Omron CX-Programmer project NewProject (CX-Programmer 9.73)

# PLC PLCMIX: CP1H XA

## Global symbols (name address type ; comment)
0.05 BOOL  ; PROXB
0.06 BOOL  ; PROXU
0.07 BOOL  ; PROXD
100.00 BOOL  ; WATER PUMP
100.01 BOOL  ; OIL PUMP
100.02 BOOL  ; VACUUM PUMP
100.03 BOOL  ; VACUUM RELEASE
100.04 BOOL  ; WATER HEATER
100.05 BOOL  ; VALVE UP
100.06 BOOL  ; VALVE DOWN
100.07 BOOL  ; UP MAX
100.08 BOOL  ; DOWN MAX
100.09 BOOL  ; POS BOWL
100.10 BOOL  ; UPPER LIMIT
100.11 BOOL  ; A
100.12 BOOL  ; UNDER LIMIT
100.13 BOOL  ; B
100.14 BOOL  ; ALARM WT TEMP
100.15 BOOL  ; ALARM MT TEMP
101.00 BOOL  ; CW
101.01 BOOL  ; CCW
101.02 BOOL  ; MAIN TIMER
101.03 BOOL  ; VALVE CW
101.04 BOOL  ; VALVE CCW
101.05 BOOL  ; ALARM LP
101.06 BOOL  ; DATA LOG
101.07 BOOL  ; ALARM TOR
10.00 BOOL  ; FLAG CALCULATE
200 CHANNEL  ; OPRESS
201 CHANNEL  ; VPRESS
2013 CHANNEL  ; RWT RAW VALUE
2014 CHANNEL  ; RWT RAW VALUE
2023 CHANNEL  ; ROT RAW VALUE
210 CHANNEL  ; DA FREQUENCY
300 CHANNEL  ; TIMER CW
301 CHANNEL  ; TIMER CCW
302 CHANNEL  ; MAIN TIMER
50.00 BOOL  ; UNDER LIMIT OPRESS
50.01 BOOL  ; UPPER LIMIT OPRESS
50.02 BOOL  ; UNDER LIMIT VPRESS
50.03 BOOL  ; UPPER LIMIT VPRESS
C0000 BOOL  ; COUNTER 1 WP
C0001 BOOL  ; COUNTER 2 WP
C0002 BOOL  ; COUNTER 1 OP
C0003 BOOL  ; COUNTER 2 OP
C0004 BOOL  ; COUNTER 1 VP
C0005 BOOL  ; COUNTER 2 VP
C0006 BOOL  ; COUNTER 1 WH
C0007 BOOL  ; COUNTER 2 WH
C0008 BOOL  ; Counter 1 UP
C0009 BOOL  ; Counter 2 UP
C0010 BOOL  ; Counter 1 DOWN
C0011 BOOL  ; Counter 2 DOWN
D0 CHANNEL  ; VALUE DA FREQUENCY
D1 CHANNEL  ; TOTAL BIT DA FREQUENCY
D10 CHANNEL  ; RWT MOV TO D10
D100 CHANNEL  ; INPUT SET MINUTE MTIM
D101 CHANNEL  ; MINUTE MTIM
D102 CHANNEL  ; INPUT SET SECOND MTIM
D103 CHANNEL  ; SECOND MTIM
D104 CHANNEL  ; INPUT SET MINUTE DIRTIM
D105 CHANNEL  ; MINUTE DIRTIM
D106 CHANNEL  ; INPUT SET SECOND DIRTIM
D107 CHANNEL  ; SECOND DIRITM
D11 CHANNEL  ; RMT MOV TO D11
D110 CHANNEL  ; MINUTE TO SECOND MTIM
D112 CHANNEL  ; SECOND TO SECOND MTIM
D114 CHANNEL  ; TOTAL SECOND MTIM
D116 CHANNEL  ; MINUTE TO SECOND DIRTIM
D118 CHANNEL  ; SECOND TO SECOND DIRTIM
D12 CHANNEL  ; ROT MOV TO D12
D120 CHANNEL  ; TOTAL SECOND DIRTIM
D130 CHANNEL  ; PV TIMER CW
D132 CHANNEL  ; PV TIMER CCW
D134 CHANNEL  ; PV MAIN TIMER
D136 CHANNEL  ; REAL SECOND
D140 CHANNEL  ; SECOND BCD TO CLOCK
D142 CHANNEL  ; SECOND DISPLAY
D144 CHANNEL  ; MINUTE DISPLAY
D146 CHANNEL  ; SET LP
D148 CHANNEL  ; DIVISOR KPA TO MPA
D150 CHANNEL  ; CONSTANTA PRES TO TORQUE
D152 CHANNEL  ; OPRESS KPA TO MPA
D154 CHANNEL  ; TORQUE RTOR NM
D156 CHANNEL  ; BACK TO NULL
D158 CHANNEL  ; SET TOR
D20 CHANNEL  ; RWT REAL NUM
D22 CHANNEL  ; RMT REAL NUM
D24 CHANNEL  ; ROT REAL NUM
D26 CHANNEL  ; DIVISOR WORD
D30 CHANNEL  ; RWT TEMP
D32 CHANNEL  ; RMT TEMP
D34 CHANNEL  ; ROT TEMP
D40 CHANNEL  ; SET WT TEMP
D42 CHANNEL  ; SET MT TEMP
D50 CHANNEL  ; RAW AD OPRESS
D51 CHANNEL  ; RAW AD VPRESS
D52 CHANNEL  ; MIN RANGE PRESSURE OPRESS
D54 CHANNEL  ; MAX RANGE PRESSURE OPRESS
D55 CHANNEL  ; MAX RANGE BIT
D56 CHANNEL  ; RESULTS SCL OPRESS
D57 CHANNEL  ; BIN OPRESS
D60 CHANNEL  ; MIN RANGE PRESSURE VPRESS
D62 CHANNEL  ; MAX RANGE PRESSURE VPRESS
D63 CHANNEL  ; MAX RANGE BIT
D64 CHANNEL  ; RESULTS SCL VPRESS
D65 CHANNEL  ; BIN VPRESS
D66 CHANNEL  ; DIVISOR 10
D68 CHANNEL  ; FLT OPRESS
D70 CHANNEL  ; FLT VPRESS
D72 CHANNEL  ; OPRESS (BAR UNIT)
D74 CHANNEL  ; BAR TO KPA
D76 CHANNEL  ; OPRESS (KPA UNIT)
D80 CHANNEL  ; MULTIPLY MBAR TO KPA
D82 CHANNEL  ; VPRESS (MBAR UNIT)
D84 CHANNEL  ; VPRESS (KPA UNIT)
D86 CHANNEL  ; PV ENCODER
D88 CHANNEL  ; FLT PV ENCODER
D90 CHANNEL  ; FLT MULTIPLY 60
D92 CHANNEL  ; FLT DIVISOR 2000
D94 CHANNEL  ; PV ENCODER MULTIPLY 60
D96 CHANNEL  ; RPM
W0.00 BOOL  ; PB WP
W0.01 BOOL  ; PB OP
W0.02 BOOL  ; PB VP
W0.03 BOOL  ; PB VR
W0.04 BOOL  ; PB WH
W0.05 BOOL  ; PB UP
W0.06 BOOL  ; PB DOWN
W0.07 BOOL  ; PB FAST
W0.08 BOOL  ; PB SLOW
W0.09 BOOL  ; SET TIME
W0.10 BOOL  ; CW
W0.11 BOOL  ; CCW
W0.12 BOOL  ; PROSES
W0.13 BOOL  ; STOP

## Program NewProgram1 (cyclic task 0)

### Section Section1

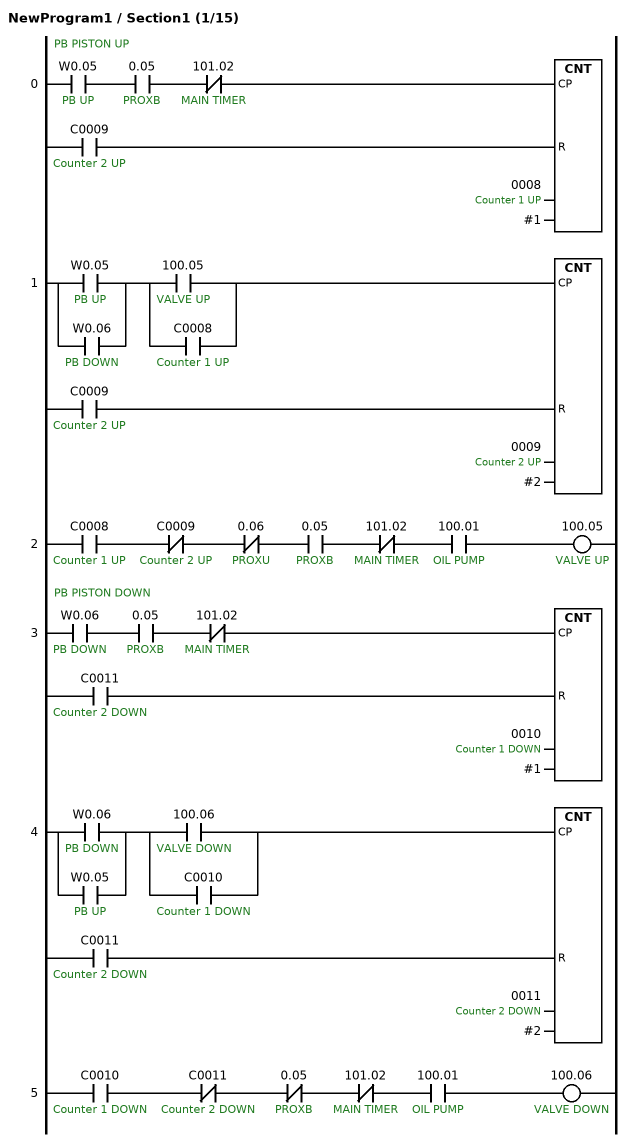
; rung 0: PB PISTON UP
LD W0.05  ; PB UP
AND 0.05  ; PROXB
ANDNOT 101.02  ; MAIN TIMER
LD C0009  ; Counter 2 UP
CNT 0008 #1  ; Counter 1 UP
; rung 1
LD W0.05  ; PB UP
OR W0.06  ; PB DOWN
LD 100.05  ; VALVE UP
OR C0008  ; Counter 1 UP
ANDLD
LD C0009  ; Counter 2 UP
CNT 0009 #2  ; Counter 2 UP
; rung 2
LD C0008  ; Counter 1 UP
ANDNOT C0009  ; Counter 2 UP
ANDNOT 0.06  ; PROXU
AND 0.05  ; PROXB
ANDNOT 101.02  ; MAIN TIMER
AND 100.01  ; OIL PUMP
OUT 100.05  ; VALVE UP
; rung 3: PB PISTON DOWN
LD W0.06  ; PB DOWN
AND 0.05  ; PROXB
ANDNOT 101.02  ; MAIN TIMER
LD C0011  ; Counter 2 DOWN
CNT 0010 #1  ; Counter 1 DOWN
; rung 4
LD W0.06  ; PB DOWN
OR W0.05  ; PB UP
LD 100.06  ; VALVE DOWN
OR C0010  ; Counter 1 DOWN
ANDLD
LD C0011  ; Counter 2 DOWN
CNT 0011 #2  ; Counter 2 DOWN
; rung 5
LD C0010  ; Counter 1 DOWN
ANDNOT C0011  ; Counter 2 DOWN
ANDNOT 0.05  ; PROXB
ANDNOT 101.02  ; MAIN TIMER
AND 100.01  ; OIL PUMP
OUT 100.06  ; VALVE DOWN

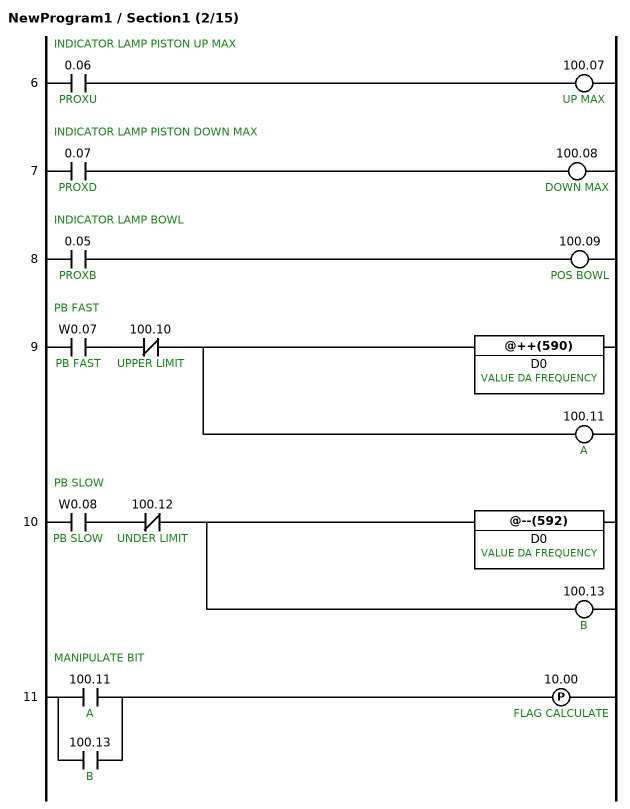
; rung 6: INDICATOR LAMP PISTON UP MAX
LD 0.06  ; PROXU
OUT 100.07  ; UP MAX
; rung 7: INDICATOR LAMP PISTON DOWN MAX
LD 0.07  ; PROXD
OUT 100.08  ; DOWN MAX
; rung 8: INDICATOR LAMP BOWL
LD 0.05  ; PROXB
OUT 100.09  ; POS BOWL
; rung 9: PB FAST
LD W0.07  ; PB FAST
ANDNOT 100.10  ; UPPER LIMIT
@++(590) D0  ; VALUE DA FREQUENCY
OUT 100.11  ; A
; rung 10: PB SLOW
LD W0.08  ; PB SLOW
ANDNOT 100.12  ; UNDER LIMIT
@--(592) D0  ; VALUE DA FREQUENCY
OUT 100.13  ; B
; rung 11: MANIPULATE BIT
LD 100.11  ; A
OR 100.13  ; B
DIFU(013) 10.00  ; FLAG CALCULATE

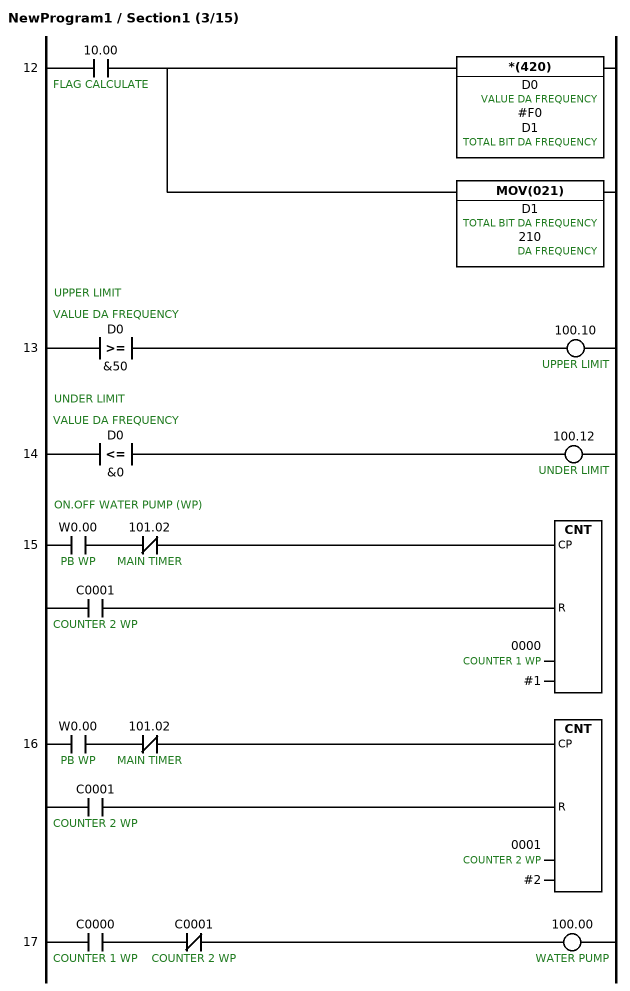
; rung 12
LD 10.00  ; FLAG CALCULATE
*(420) D0 #F0 D1  ; VALUE DA FREQUENCY, TOTAL BIT DA FREQUENCY
MOV(021) D1 210  ; TOTAL BIT DA FREQUENCY, DA FREQUENCY
; rung 13: UPPER LIMIT
LD>=(325) D0 &50  ; VALUE DA FREQUENCY
OUT 100.10  ; UPPER LIMIT
; rung 14: UNDER LIMIT
LD<=(315) D0 &0  ; VALUE DA FREQUENCY
OUT 100.12  ; UNDER LIMIT
; rung 15: ON.OFF WATER PUMP (WP)
LD W0.00  ; PB WP
ANDNOT 101.02  ; MAIN TIMER
LD C0001  ; COUNTER 2 WP
CNT 0000 #1  ; COUNTER 1 WP
; rung 16
LD W0.00  ; PB WP
ANDNOT 101.02  ; MAIN TIMER
LD C0001  ; COUNTER 2 WP
CNT 0001 #2  ; COUNTER 2 WP
; rung 17
LD C0000  ; COUNTER 1 WP
ANDNOT C0001  ; COUNTER 2 WP
OUT 100.00  ; WATER PUMP

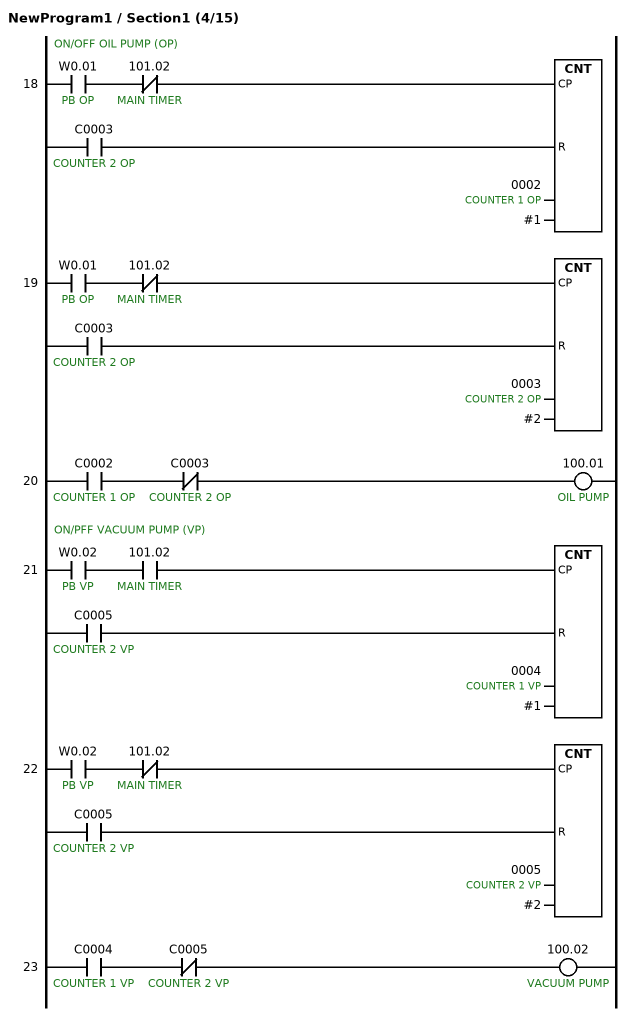
; rung 18: ON/OFF OIL PUMP (OP)
LD W0.01  ; PB OP
ANDNOT 101.02  ; MAIN TIMER
LD C0003  ; COUNTER 2 OP
CNT 0002 #1  ; COUNTER 1 OP
; rung 19
LD W0.01  ; PB OP
ANDNOT 101.02  ; MAIN TIMER
LD C0003  ; COUNTER 2 OP
CNT 0003 #2  ; COUNTER 2 OP
; rung 20
LD C0002  ; COUNTER 1 OP
ANDNOT C0003  ; COUNTER 2 OP
OUT 100.01  ; OIL PUMP
; rung 21: ON/PFF VACUUM PUMP (VP)
LD W0.02  ; PB VP
AND 101.02  ; MAIN TIMER
LD C0005  ; COUNTER 2 VP
CNT 0004 #1  ; COUNTER 1 VP
; rung 22
LD W0.02  ; PB VP
ANDNOT 101.02  ; MAIN TIMER
LD C0005  ; COUNTER 2 VP
CNT 0005 #2  ; COUNTER 2 VP
; rung 23
LD C0004  ; COUNTER 1 VP
ANDNOT C0005  ; COUNTER 2 VP
OUT 100.02  ; VACUUM PUMP

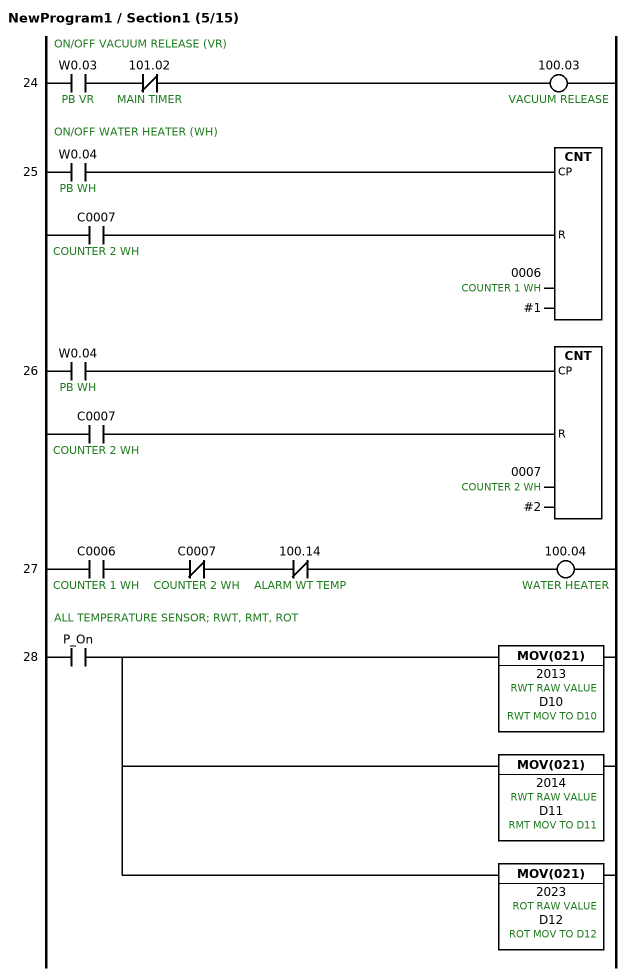
; rung 24: ON/OFF VACUUM RELEASE (VR)
LD W0.03  ; PB VR
ANDNOT 101.02  ; MAIN TIMER
OUT 100.03  ; VACUUM RELEASE
; rung 25: ON/OFF WATER HEATER (WH)
LD W0.04  ; PB WH
LD C0007  ; COUNTER 2 WH
CNT 0006 #1  ; COUNTER 1 WH
; rung 26
LD W0.04  ; PB WH
LD C0007  ; COUNTER 2 WH
CNT 0007 #2  ; COUNTER 2 WH
; rung 27
LD C0006  ; COUNTER 1 WH
ANDNOT C0007  ; COUNTER 2 WH
ANDNOT 100.14  ; ALARM WT TEMP
OUT 100.04  ; WATER HEATER
; rung 28: ALL TEMPERATURE SENSOR; RWT, RMT, ROT
LD P_On
MOV(021) 2013 D10  ; RWT RAW VALUE, RWT MOV TO D10
MOV(021) 2014 D11  ; RWT RAW VALUE, RMT MOV TO D11
MOV(021) 2023 D12  ; ROT RAW VALUE, ROT MOV TO D12

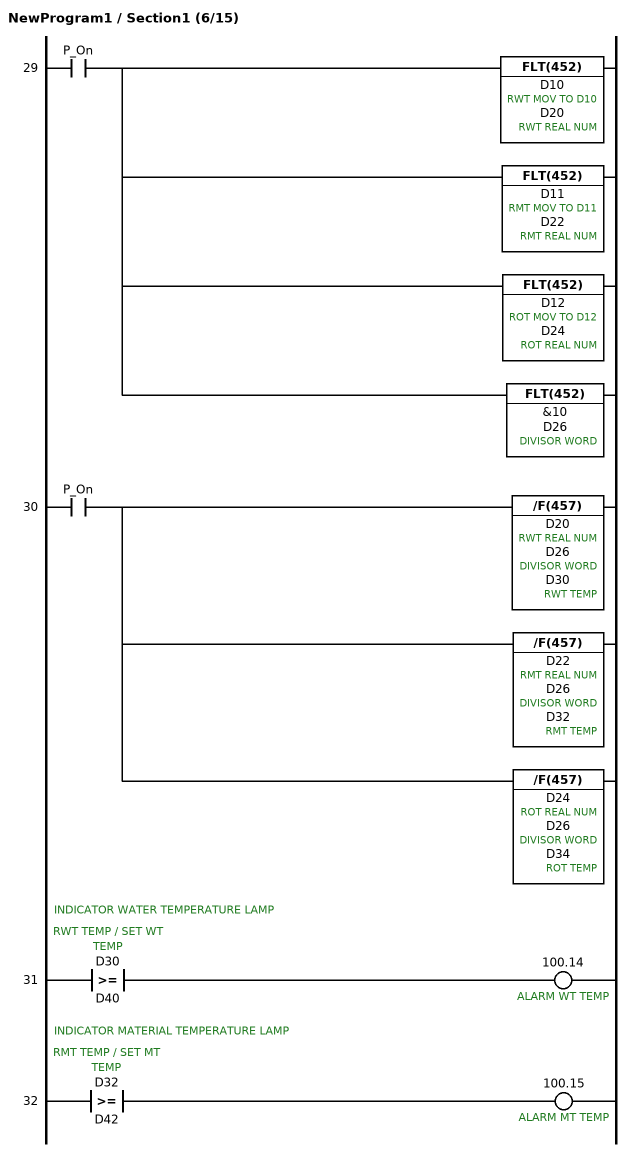
; rung 29
LD P_On
FLT(452) D10 D20  ; RWT MOV TO D10, RWT REAL NUM
FLT(452) D11 D22  ; RMT MOV TO D11, RMT REAL NUM
FLT(452) D12 D24  ; ROT MOV TO D12, ROT REAL NUM
FLT(452) &10 D26  ; DIVISOR WORD
; rung 30
LD P_On
/F(457) D20 D26 D30  ; RWT REAL NUM, DIVISOR WORD, RWT TEMP
/F(457) D22 D26 D32  ; RMT REAL NUM, DIVISOR WORD, RMT TEMP
/F(457) D24 D26 D34  ; ROT REAL NUM, DIVISOR WORD, ROT TEMP
; rung 31: INDICATOR WATER TEMPERATURE LAMP
LD>=F(334) D30 D40  ; RWT TEMP, SET WT TEMP
OUT 100.14  ; ALARM WT TEMP
; rung 32: INDICATOR MATERIAL TEMPERATURE LAMP
LD>=F(334) D32 D42  ; RMT TEMP, SET MT TEMP
OUT 100.15  ; ALARM MT TEMP

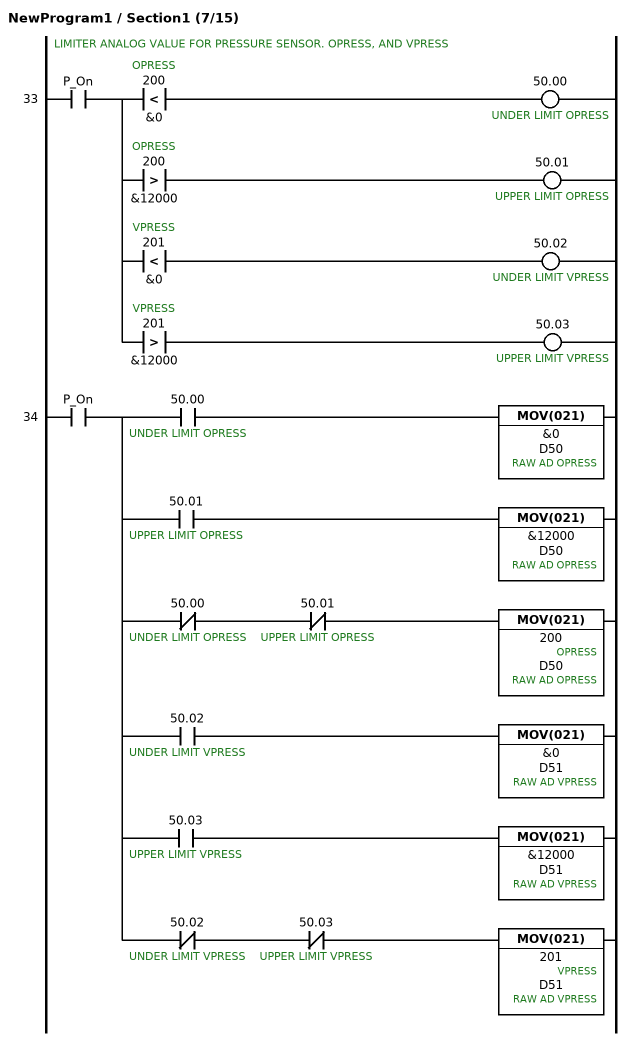
; rung 33: LIMITER ANALOG VALUE FOR PRESSURE SENSOR. OPRESS, AND VPRESS
LD P_On
OUT TR0
AND<S(312) 200 &0  ; OPRESS
OUT 50.00  ; UNDER LIMIT OPRESS
LD TR0
AND>S(322) 200 &12000  ; OPRESS
OUT 50.01  ; UPPER LIMIT OPRESS
LD TR0
AND<S(312) 201 &0  ; VPRESS
OUT 50.02  ; UNDER LIMIT VPRESS
LD TR0
AND>S(322) 201 &12000  ; VPRESS
OUT 50.03  ; UPPER LIMIT VPRESS
; rung 34
LD P_On
OUT TR0
AND 50.00  ; UNDER LIMIT OPRESS
MOV(021) &0 D50  ; RAW AD OPRESS
LD TR0
AND 50.01  ; UPPER LIMIT OPRESS
MOV(021) &12000 D50  ; RAW AD OPRESS
LD TR0
ANDNOT 50.00  ; UNDER LIMIT OPRESS
ANDNOT 50.01  ; UPPER LIMIT OPRESS
MOV(021) 200 D50  ; OPRESS, RAW AD OPRESS
LD TR0
AND 50.02  ; UNDER LIMIT VPRESS
MOV(021) &0 D51  ; RAW AD VPRESS
LD TR0
AND 50.03  ; UPPER LIMIT VPRESS
MOV(021) &12000 D51  ; RAW AD VPRESS
LD TR0
ANDNOT 50.02  ; UNDER LIMIT VPRESS
ANDNOT 50.03  ; UPPER LIMIT VPRESS
MOV(021) 201 D51  ; VPRESS, RAW AD VPRESS

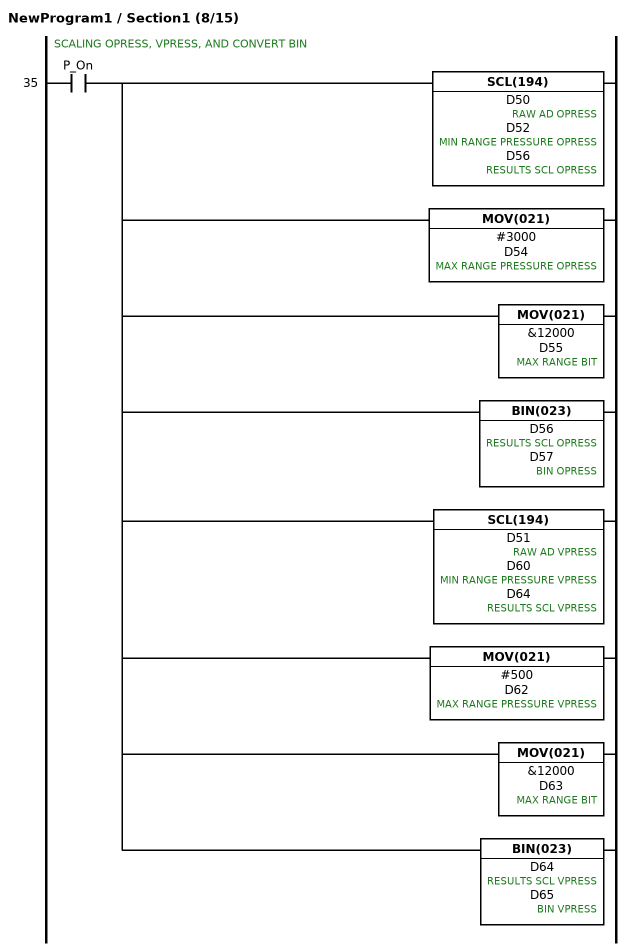
; rung 35: SCALING OPRESS, VPRESS, AND CONVERT BIN
LD P_On
SCL(194) D50 D52 D56  ; RAW AD OPRESS, MIN RANGE PRESSURE OPRESS, RESULTS SCL OPRESS
MOV(021) #3000 D54  ; MAX RANGE PRESSURE OPRESS
MOV(021) &12000 D55  ; MAX RANGE BIT
BIN(023) D56 D57  ; RESULTS SCL OPRESS, BIN OPRESS
SCL(194) D51 D60 D64  ; RAW AD VPRESS, MIN RANGE PRESSURE VPRESS, RESULTS SCL VPRESS
MOV(021) #500 D62  ; MAX RANGE PRESSURE VPRESS
MOV(021) &12000 D63  ; MAX RANGE BIT
BIN(023) D64 D65  ; RESULTS SCL VPRESS, BIN VPRESS

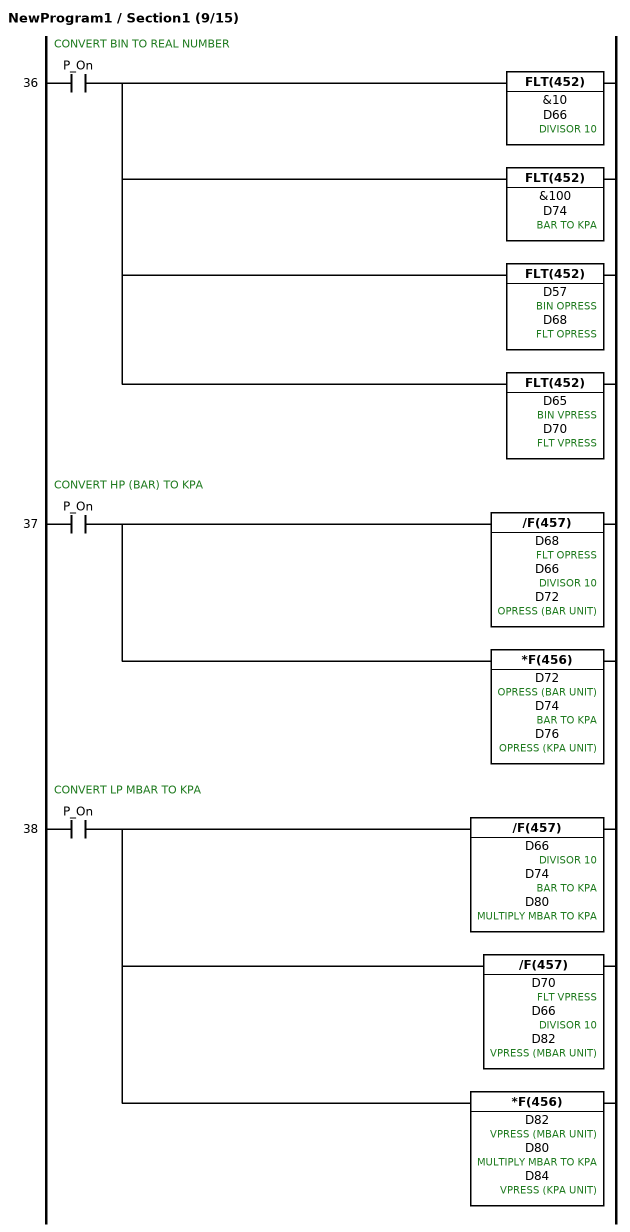
; rung 36: CONVERT BIN TO REAL NUMBER
LD P_On
FLT(452) &10 D66  ; DIVISOR 10
FLT(452) &100 D74  ; BAR TO KPA
FLT(452) D57 D68  ; BIN OPRESS, FLT OPRESS
FLT(452) D65 D70  ; BIN VPRESS, FLT VPRESS
; rung 37: CONVERT HP (BAR) TO KPA
LD P_On
/F(457) D68 D66 D72  ; FLT OPRESS, DIVISOR 10, OPRESS (BAR UNIT)
*F(456) D72 D74 D76  ; OPRESS (BAR UNIT), BAR TO KPA, OPRESS (KPA UNIT)
; rung 38: CONVERT LP MBAR TO KPA
LD P_On
/F(457) D66 D74 D80  ; DIVISOR 10, BAR TO KPA, MULTIPLY MBAR TO KPA
/F(457) D70 D66 D82  ; FLT VPRESS, DIVISOR 10, VPRESS (MBAR UNIT)
*F(456) D82 D80 D84  ; VPRESS (MBAR UNIT), MULTIPLY MBAR TO KPA, VPRESS (KPA UNIT)

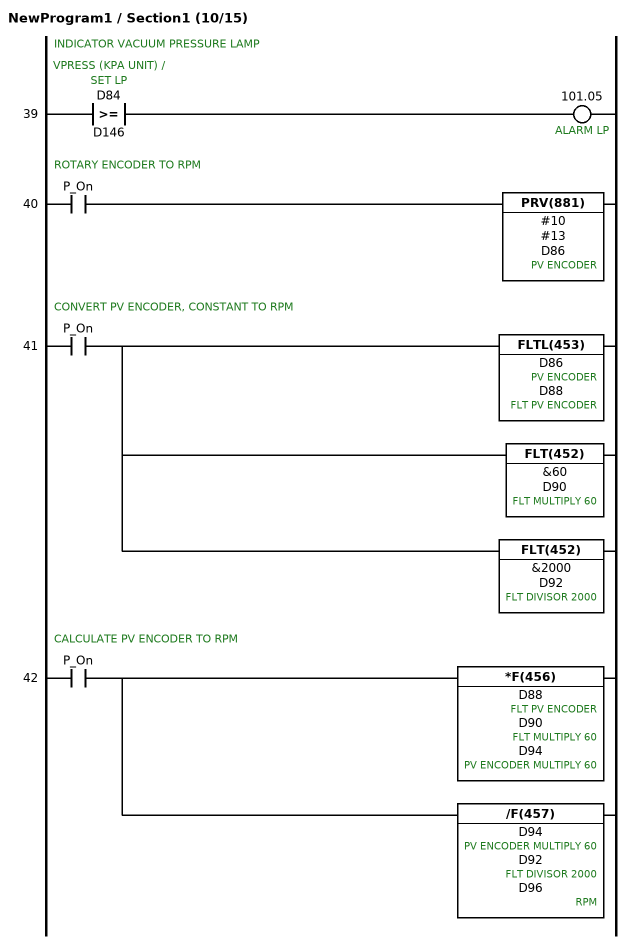
; rung 39: INDICATOR VACUUM PRESSURE LAMP
LD>=F(334) D84 D146  ; VPRESS (KPA UNIT), SET LP
OUT 101.05  ; ALARM LP
; rung 40: ROTARY ENCODER TO RPM
LD P_On
PRV(881) #10 #13 D86  ; PV ENCODER
; rung 41: CONVERT PV ENCODER, CONSTANT TO RPM
LD P_On
FLTL(453) D86 D88  ; PV ENCODER, FLT PV ENCODER
FLT(452) &60 D90  ; FLT MULTIPLY 60
FLT(452) &2000 D92  ; FLT DIVISOR 2000
; rung 42: CALCULATE PV ENCODER TO RPM
LD P_On
*F(456) D88 D90 D94  ; FLT PV ENCODER, FLT MULTIPLY 60, PV ENCODER MULTIPLY 60
/F(457) D94 D92 D96  ; PV ENCODER MULTIPLY 60, FLT DIVISOR 2000, RPM

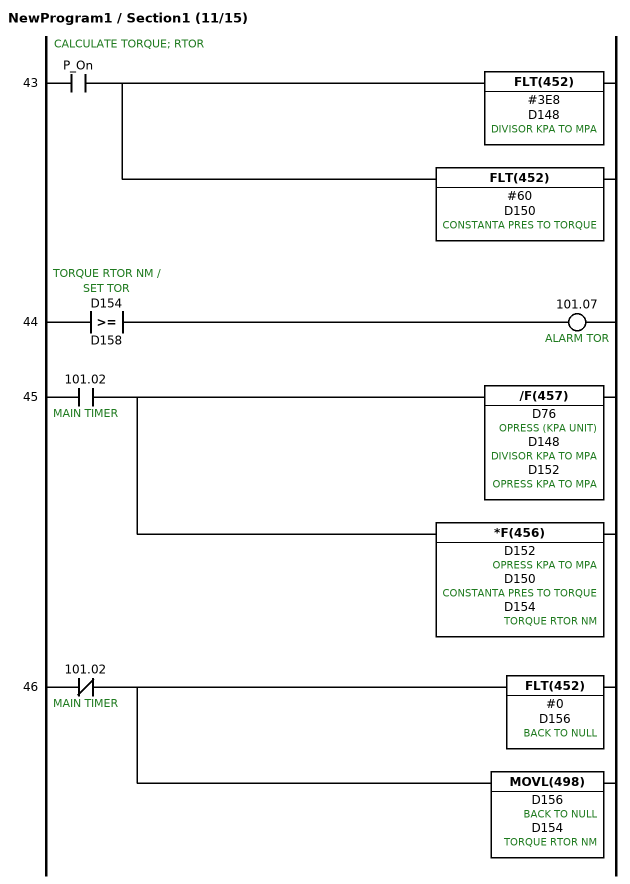
; rung 43: CALCULATE TORQUE; RTOR
LD P_On
FLT(452) #3E8 D148  ; DIVISOR KPA TO MPA
FLT(452) #60 D150  ; CONSTANTA PRES TO TORQUE
; rung 44
LD>=F(334) D154 D158  ; TORQUE RTOR NM, SET TOR
OUT 101.07  ; ALARM TOR
; rung 45
LD 101.02  ; MAIN TIMER
/F(457) D76 D148 D152  ; OPRESS (KPA UNIT), DIVISOR KPA TO MPA, OPRESS KPA TO MPA
*F(456) D152 D150 D154  ; OPRESS KPA TO MPA, CONSTANTA PRES TO TORQUE, TORQUE RTOR NM
; rung 46
LDNOT 101.02  ; MAIN TIMER
FLT(452) #0 D156  ; BACK TO NULL
MOVL(498) D156 D154  ; BACK TO NULL, TORQUE RTOR NM

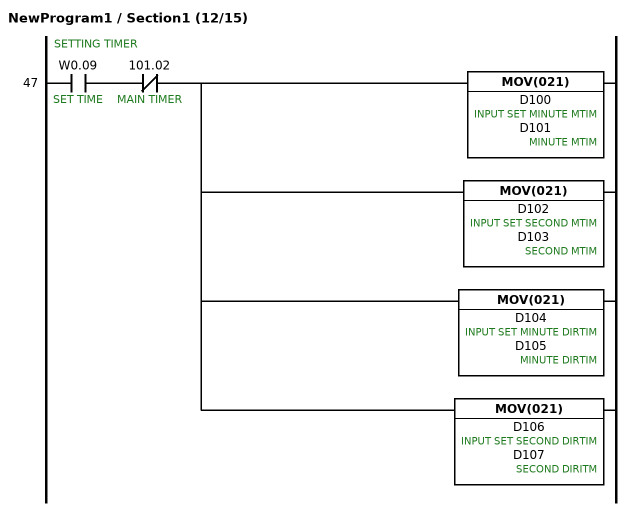
; rung 47: SETTING TIMER
LD W0.09  ; SET TIME
ANDNOT 101.02  ; MAIN TIMER
MOV(021) D100 D101  ; INPUT SET MINUTE MTIM, MINUTE MTIM
MOV(021) D102 D103  ; INPUT SET SECOND MTIM, SECOND MTIM
MOV(021) D104 D105  ; INPUT SET MINUTE DIRTIM, MINUTE DIRTIM
MOV(021) D106 D107  ; INPUT SET SECOND DIRTIM, SECOND DIRITM

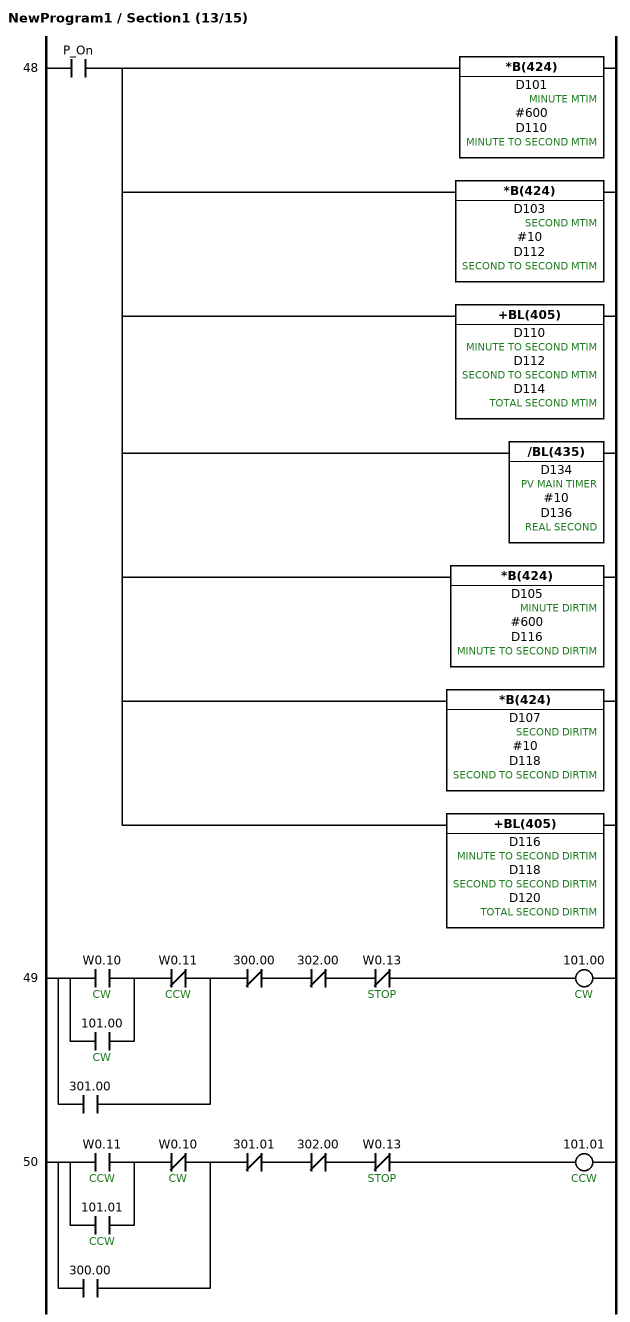
; rung 48
LD P_On
*B(424) D101 #600 D110  ; MINUTE MTIM, MINUTE TO SECOND MTIM
*B(424) D103 #10 D112  ; SECOND MTIM, SECOND TO SECOND MTIM
+BL(405) D110 D112 D114  ; MINUTE TO SECOND MTIM, SECOND TO SECOND MTIM, TOTAL SECOND MTIM
/BL(435) D134 #10 D136  ; PV MAIN TIMER, REAL SECOND
*B(424) D105 #600 D116  ; MINUTE DIRTIM, MINUTE TO SECOND DIRTIM
*B(424) D107 #10 D118  ; SECOND DIRITM, SECOND TO SECOND DIRTIM
+BL(405) D116 D118 D120  ; MINUTE TO SECOND DIRTIM, SECOND TO SECOND DIRTIM, TOTAL SECOND DIRTIM
; rung 49
LD W0.10  ; CW
OR 101.00  ; CW
ANDNOT W0.11  ; CCW
OR 301.00
ANDNOT 300.00
ANDNOT 302.00
ANDNOT W0.13  ; STOP
OUT 101.00  ; CW
; rung 50
LD W0.11  ; CCW
OR 101.01  ; CCW
ANDNOT W0.10  ; CW
OR 300.00
ANDNOT 301.01
ANDNOT 302.00
ANDNOT W0.13  ; STOP
OUT 101.01  ; CCW

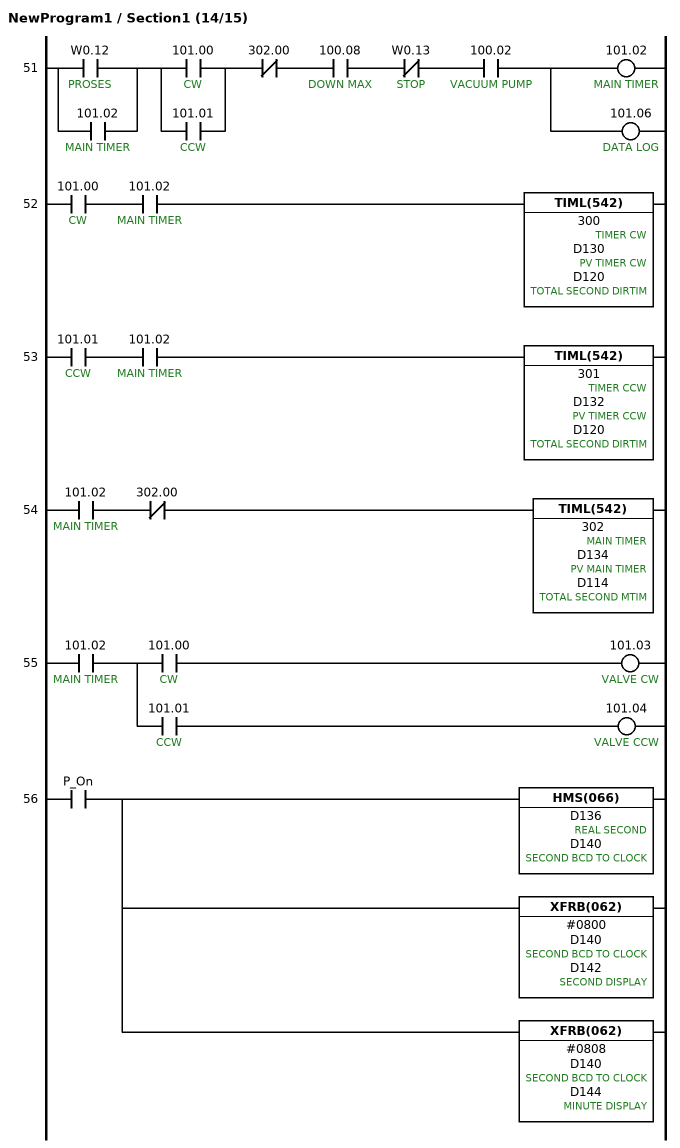
; rung 51
LD W0.12  ; PROSES
OR 101.02  ; MAIN TIMER
LD 101.00  ; CW
OR 101.01  ; CCW
ANDLD
ANDNOT 302.00
AND 100.08  ; DOWN MAX
ANDNOT W0.13  ; STOP
AND 100.02  ; VACUUM PUMP
OUT 101.02  ; MAIN TIMER
OUT 101.06  ; DATA LOG
; rung 52
LD 101.00  ; CW
AND 101.02  ; MAIN TIMER
TIML(542) 300 D130 D120  ; TIMER CW, PV TIMER CW, TOTAL SECOND DIRTIM
; rung 53
LD 101.01  ; CCW
AND 101.02  ; MAIN TIMER
TIML(542) 301 D132 D120  ; TIMER CCW, PV TIMER CCW, TOTAL SECOND DIRTIM
; rung 54
LD 101.02  ; MAIN TIMER
ANDNOT 302.00
TIML(542) 302 D134 D114  ; MAIN TIMER, PV MAIN TIMER, TOTAL SECOND MTIM
; rung 55
LD 101.02  ; MAIN TIMER
OUT TR0
AND 101.00  ; CW
OUT 101.03  ; VALVE CW
LD TR0
AND 101.01  ; CCW
OUT 101.04  ; VALVE CCW
; rung 56
LD P_On
HMS(066) D136 D140  ; REAL SECOND, SECOND BCD TO CLOCK
XFRB(062) #0800 D140 D142  ; SECOND BCD TO CLOCK, SECOND DISPLAY
XFRB(062) #0808 D140 D144  ; SECOND BCD TO CLOCK, MINUTE DISPLAY

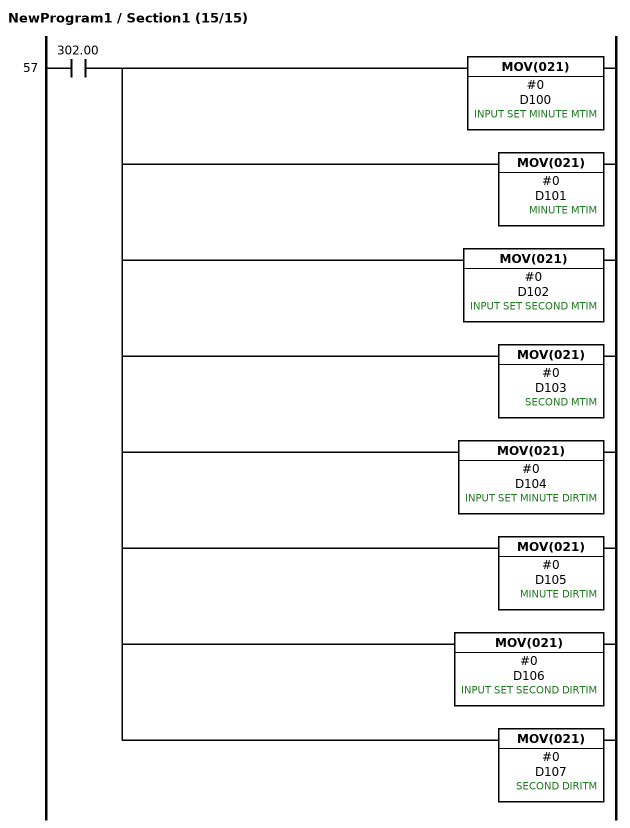
; rung 57
LD 302.00
MOV(021) #0 D100  ; INPUT SET MINUTE MTIM
MOV(021) #0 D101  ; MINUTE MTIM
MOV(021) #0 D102  ; INPUT SET SECOND MTIM
MOV(021) #0 D103  ; SECOND MTIM
MOV(021) #0 D104  ; INPUT SET MINUTE DIRTIM
MOV(021) #0 D105  ; MINUTE DIRTIM
MOV(021) #0 D106  ; INPUT SET SECOND DIRTIM
MOV(021) #0 D107  ; SECOND DIRITM

### Section END
; rung 0
END(001)